(* IEC 61131-3 sources: MotionTestBenchMaster/Logical/30_MC/Libraries/MotionLib/FB, 9 files *)

(* ---- FB_AbsolutePosCalculation.st ---- *)
FUNCTION_BLOCK FB_AbsolutePosCalculation
	IF i_xEnable THEN

		IF NOT i_pstAxis.iq_stStatus.q_stMainAxisStatus.q_xInitDone OR i_pstAxis.iq_stStatus.q_stMainAxisStatus.q_xError THEN
			xPositionValid 		:= FALSE;
		ELSIF i_xPositionSensor AND NOT xPositionValid THEN
			lrAbsolutePosition 	:= i_pstAxis.iq_stStatus.q_stMainAxisStatus.q_lrPosition + 360.0 * MAX((i_uiAbsolutePositionOffset - 1), 0);
			xPositionValid 		:= TRUE;
			lrOldPosition 		:= i_pstAxis.iq_stStatus.q_stMainAxisStatus.q_lrPosition;
		ELSE
			lrIncrement			:= i_pstAxis.iq_stStatus.q_stMainAxisStatus.q_lrPosition - lrOldPosition;

			IF lrIncrement < -180.0 THEN
				lrIncrement := lrIncrement + 360.0;
			ELSIF lrIncrement > 180.0 THEN
				lrIncrement := lrIncrement - 360.0;
			END_IF

			lrAbsolutePosition	:= lrAbsolutePosition + lrIncrement;
			lrOldPosition		:= i_pstAxis.iq_stStatus.q_stMainAxisStatus.q_lrPosition;
		END_IF

		lrAbsolutePosition		:= FC_LongRealReminder(lrAbsolutePosition, 360.0 * i_uiStepsNumber, 0);

		q_xPositionValid		:= xPositionValid;
		q_lrAbsolutePosition	:= lrAbsolutePosition;
	END_IF
END_FUNCTION_BLOCK

(* ---- FB_CamGenerator.st ---- *)
(* Cam Generator Function Block *)
FUNCTION_BLOCK FB_CamGenerator
	IF i_xEnable AND i_usiNumberOfPulse > 0 THEN
		IF i_usiNumberOfPulse = 1 AND i_rOnPosition <> i_rOffPosition THEN
			rAdvPosition		:= i_rAdvanceTime * i_prAxisVelocity / 1000.0;
			q_xAdvError			:= (ABS(rAdvPosition) >= 360);

			i_pxPointerStepAdv	:= ((i_rOnPosition - rAdvPosition) < 0);

			rOnPositionA		:= FC_RealReminder(i_rOnPosition - rAdvPosition,	360.0, 0);
			rOffPositionA		:= FC_RealReminder(i_rOffPosition - rAdvPosition,	360.0, 0);

			(* CAM A GENERATION *)
			IF(rOnPositionA < rOffPositionA) THEN
				xCamValueA	:= (i_plrAxisPosition >= rOnPositionA) AND (i_plrAxisPosition < rOffPositionA);
			ELSE
				xCamValueA	:= i_plrAxisPosition >= rOnPositionA OR i_plrAxisPosition < rOffPositionA;
			END_IF

			IF xCamValueA <> xOldCamValueA THEN
				rTempReal	:= SEL(xCamValueA, rOffPositionA, rOnPositionA);
				rTempReal	:= rTempReal - LREAL_TO_REAL(i_plrAxisPosition);
				IF ABS(rTempReal) > 0.5 AND ABS(rTempReal) < 359.5 THEN
					xOldCamValueA := xCamValueA;
				END_IF
			END_IF

			(* CAM B GENERATION *)
			IF i_rOnPositionB <> 0 AND i_rOffPositionB <> 0 THEN
				rOnPositionB		:= FC_RealReminder(i_rOnPositionB - rAdvPosition,	360.0, 0);
				rOffPositionB		:= FC_RealReminder(i_rOffPositionB - rAdvPosition,	360.0, 0);
				IF(rOnPositionB < rOffPositionB) THEN
					xCamValueB	:= (i_plrAxisPosition >= rOnPositionB) AND (i_plrAxisPosition < rOffPositionB);
				ELSE
					xCamValueB	:= i_plrAxisPosition >= rOnPositionB OR i_plrAxisPosition < rOffPositionB;
				END_IF

				IF xCamValueB <> xOldCamValueB THEN
					rTempReal	:= SEL(xCamValueB, rOffPositionB, rOnPositionB);
					rTempReal	:= rTempReal - LREAL_TO_REAL(i_plrAxisPosition);
					IF ABS(rTempReal) > 0.5 AND ABS(rTempReal) < 359.5 THEN
						xOldCamValueB	:=	xCamValueB;
					END_IF
				END_IF

				(* Debounce *)
				CASE usiStep OF
					0:(* INIT *)
						usiStep := 100;

					100:(* WAIT FOR CAM A RAISING EDGE *)
						IF xCamValueA THEN
							i_pxPointerOutput := TRUE;
							usiStep := 110;
						END_IF

					110:(* WAIT FOR CAM B FALLING EDGE *)
						IF NOT xCamValueB THEN
							usiStep := 120;
						END_IF

					120:(*  WAIT FOR CAM A FALLING EDGE *)
						IF NOT xCamValueA THEN
							i_pxPointerOutput := FALSE;
							usiStep := 130;
						END_IF

					130:(* WAIT FOR CAM B RAISING EDGE *)
						IF xCamValueB THEN
							usiStep := 100;
						END_IF

					ELSE
						usiStep := 200;
				END_CASE
			ELSE
				(* Simple cam A generator *)
				i_pxPointerOutput	:= xOldCamValueA;
			END_IF
		ELSIF i_usiNumberOfPulse <= 10 THEN
			i_pxPointerStepAdv	:= FALSE;
			i_pxPointerOutput	:= FC_RealReminder(LREAL_TO_REAL(i_plrAxisPosition), 360.0 / i_usiNumberOfPulse, 0) >= 180.0 / i_usiNumberOfPulse;
		END_IF
	ELSE
		i_pxPointerOutput	:= FALSE;
		q_xAdvError			:= FALSE;
	END_IF
END_FUNCTION_BLOCK

(* Cam Generator Function Block *)
FUNCTION_BLOCK FB_CamGenerator_v2
	IF i_xEnable AND i_usiNumberOfPulse > 0 THEN
		IF i_usiNumberOfPulse = 1 AND i_rOnPosition <> i_rOffPosition THEN
			rPosition			:= DINT_TO_REAL(i_pdiAxisPosition MOD 36000) / 100.0;
			rAdvPosition		:= i_rAdvanceTime * i_prAxisVelocity / 100000.0; //v1.4
			q_xAdvError			:= (ABS(rAdvPosition) >= 360);

			i_pxPointerStepAdv	:= ((i_rOnPosition - rAdvPosition) < 0);

			rOnPosition		:= FC_RealReminder(i_rOnPosition - rAdvPosition,	360.0, 0);
			rOffPosition	:= FC_RealReminder(i_rOffPosition - rAdvPosition,	360.0, 0);

			(* CAM GENERATION *)
			IF(rOnPosition < rOffPosition) THEN
				xCamValue	:= (rPosition >= rOnPosition) AND (rPosition < rOffPosition);
			ELSE
				xCamValue	:= rPosition >= rOnPosition OR rPosition < rOffPosition;
			END_IF

			IF xCamValue <> xOldCamValue THEN
				rTempReal	:= SEL(xCamValue, rOffPosition, rOnPosition);
				rTempReal	:= rTempReal - rPosition;
				IF ABS(rTempReal) > 0.5 AND ABS(rTempReal) < 359.5 THEN
					xOldCamValue := xCamValue;
				END_IF
			END_IF

			i_pxPointerOutput	:= xOldCamValue;
		ELSIF i_usiNumberOfPulse <= 10 THEN
			i_pxPointerStepAdv	:= FALSE;
			rPosition			:= DINT_TO_REAL(i_pdiAxisPosition MOD 36000) / 100.0;
			i_pxPointerOutput	:= FC_RealReminder(rPosition, 360.0 / i_usiNumberOfPulse, 0) >= 180.0 / i_usiNumberOfPulse;
		END_IF
	ELSE
		i_pxPointerOutput	:= FALSE;
		q_xAdvError			:= FALSE;
	END_IF
END_FUNCTION_BLOCK

(* ---- FB_CamGeneratorAB.st ---- *)
(* Cam Generator Function Block *)
FUNCTION_BLOCK FB_CamGeneratorAB
	IF i_xEnable THEN
		IF (i_rOnPositionA <> i_rOffPositionA) AND (i_rOnPositionB <> i_rOffPositionB) THEN
			rAdvPosition		:= i_rAdvanceTime * i_prAxisVelocity / 1000.0;
			q_xAdvError			:= (ABS(rAdvPosition) >= 360);

			i_pxPointerStepAdvA	:= ((i_rOnPositionA - rAdvPosition) < 0);
			i_pxPointerStepAdvB	:= ((i_rOnPositionB - rAdvPosition) < 0);

			rOnPositionA		:= FC_RealReminder(i_rOnPositionA - rAdvPosition,	360.0, 0);
			rOffPositionA		:= FC_RealReminder(i_rOffPositionA - rAdvPosition,	360.0, 0);

			rOnPositionB		:= FC_RealReminder(i_rOnPositionB - rAdvPosition,	360.0, 0);
			rOffPositionB		:= FC_RealReminder(i_rOffPositionB - rAdvPosition,	360.0, 0);

			(* CAM A GENERATION *)
			IF(rOnPositionA < rOffPositionA) THEN
				xCamValueA	:= (i_plrAxisPosition >= rOnPositionA) AND (i_plrAxisPosition < rOffPositionA);
			ELSE
				xCamValueA	:= i_plrAxisPosition >= rOnPositionA OR i_plrAxisPosition < rOffPositionA;
			END_IF

			IF xCamValueA <> xOldCamValueA THEN
				rTempReal	:= SEL(xCamValueA, rOffPositionA, rOnPositionA);
				rTempReal	:= rTempReal - LREAL_TO_REAL(i_plrAxisPosition);
				IF ABS(rTempReal) > 0.5 AND ABS(rTempReal) < 359.5 THEN
					xOldCamValueA := xCamValueA;
				END_IF
			END_IF

			(* CAM B GENERATION *)
			IF(rOnPositionB < rOffPositionB) THEN
				xCamValueB	:= (i_plrAxisPosition >= rOnPositionB) AND (i_plrAxisPosition < rOffPositionB);
			ELSE
				xCamValueB	:= i_plrAxisPosition >= rOnPositionB OR i_plrAxisPosition < rOffPositionB;
			END_IF

			IF xCamValueB <> xOldCamValueB THEN
				rTempReal	:= SEL(xCamValueB, rOffPositionB, rOnPositionB);
				rTempReal	:= rTempReal - LREAL_TO_REAL(i_plrAxisPosition);
				IF ABS(rTempReal) > 0.5 AND ABS(rTempReal) < 359.5 THEN
					xOldCamValueB	:=	xCamValueB;
				END_IF
			END_IF

			(* Debounce *)
			CASE usiStep OF
				0:(* INIT *)
					usiStep := 10;

				10:(* WAIT FIRST CAM RAISING EDGE *)
					IF rOnPositionB < rOffPositionA THEN
						IF xCamValueA THEN
							i_pxPointerOutputA := TRUE;
							usiStep := 100;
						END_IF
					ELSE
						IF xCamValueB THEN
							i_pxPointerOutputB := TRUE;
							usiStep := 200;
						END_IF
					END_IF

				100:(* WAIT CAM B RISE EDGE *)
					IF xCamValueB THEN
						i_pxPointerOutputB := TRUE;
						usiStep := 110;
					END_IF

				110:(* WAIT CAM A FALLING EDGE *)
					IF NOT xCamValueA THEN
						i_pxPointerOutputA := FALSE;
						usiStep := 120;
					END_IF

				120:(* WAIT FOR CAM B FALLING EDGE *)
					IF NOT xCamValueB THEN
						i_pxPointerOutputB := FALSE;
						usiStep := 10;
					END_IF

				200:(* WAIT CAM A RISE EDGE *)
					IF xCamValueA THEN
						i_pxPointerOutputA := TRUE;
						usiStep := 210;
					END_IF

				210:(* WAIT CAM B FALLING EDGE *)
					IF NOT xCamValueB THEN
						i_pxPointerOutputB := FALSE;
						usiStep := 220;
					END_IF

				220:(* WAIT FOR CAM A FALLING EDGE *)
					IF NOT xCamValueA THEN
						i_pxPointerOutputA := FALSE;
						usiStep := 10;
					END_IF

				ELSE
					usiStep := 255;
			END_CASE
		END_IF
	ELSE
		i_pxPointerOutputA	:= FALSE;
		i_pxPointerOutputB	:= FALSE;
		q_xAdvError			:= FALSE;
	END_IF
END_FUNCTION_BLOCK

(* Cam Generator Function Block *)
FUNCTION_BLOCK FB_CamGeneratorAB_v2
	IF i_xEnable THEN
		IF (i_rOnPositionA <> i_rOffPositionA) AND (i_rOnPositionB <> i_rOffPositionB) THEN
			rPosition			:= DINT_TO_REAL(i_pdiAxisPosition MOD 36000) / 100.0;
			rAdvPosition		:= i_rAdvanceTime * i_prAxisVelocity / 100000.0; //v1.6
			q_xAdvError			:= (ABS(rAdvPosition) >= 360);

			i_pxPointerStepAdvA	:= ((i_rOnPositionA - rAdvPosition) < 0);
			i_pxPointerStepAdvB	:= ((i_rOnPositionB - rAdvPosition) < 0);

			rOnPositionA		:= FC_RealReminder(i_rOnPositionA - rAdvPosition,	360.0, 0);
			rOffPositionA		:= FC_RealReminder(i_rOffPositionA - rAdvPosition,	360.0, 0);

			rOnPositionB		:= FC_RealReminder(i_rOnPositionB - rAdvPosition,	360.0, 0);
			rOffPositionB		:= FC_RealReminder(i_rOffPositionB - rAdvPosition,	360.0, 0);

			(* CAM A GENERATION *)
			IF(rOnPositionA < rOffPositionA) THEN
				xCamValueA	:= (rPosition >= rOnPositionA) AND (rPosition < rOffPositionA);
			ELSE
				xCamValueA	:= rPosition >= rOnPositionA OR rPosition < rOffPositionA;
			END_IF

			IF xCamValueA <> xOldCamValueA THEN
				rTempReal	:= SEL(xCamValueA, rOffPositionA, rOnPositionA);
				rTempReal	:= rTempReal - rPosition;
				IF ABS(rTempReal) > 0.5 AND ABS(rTempReal) < 359.5 THEN
					xOldCamValueA := xCamValueA;
				END_IF
			END_IF

			(* CAM B GENERATION *)
			IF(rOnPositionB < rOffPositionB) THEN
				xCamValueB	:= (rPosition >= rOnPositionB) AND (rPosition < rOffPositionB);
			ELSE
				xCamValueB	:= rPosition >= rOnPositionB OR rPosition < rOffPositionB;
			END_IF

			IF xCamValueB <> xOldCamValueB THEN
				rTempReal	:= SEL(xCamValueB, rOffPositionB, rOnPositionB);
				rTempReal	:= rTempReal - rPosition;
				IF ABS(rTempReal) > 0.5 AND ABS(rTempReal) < 359.5 THEN
					xOldCamValueB	:=	xCamValueB;
				END_IF
			END_IF

			(* Debounce *)
			CASE usiStep OF
				0:(* INIT *)
					usiStep := 10;

				10:(* WAIT FIRST CAM RAISING EDGE *)
					IF rOnPositionB < rOffPositionA THEN
						IF xCamValueA THEN
							i_pxPointerOutputA := TRUE;
							usiStep := 100;
						END_IF
					ELSE
						IF xCamValueB THEN
							i_pxPointerOutputB := TRUE;
							usiStep := 200;
						END_IF
					END_IF

				100:(* WAIT CAM B RISE EDGE *)
					IF xCamValueB THEN
						i_pxPointerOutputB := TRUE;
						usiStep := 110;
					END_IF

				110:(* WAIT CAM A FALLING EDGE *)
					IF NOT xCamValueA THEN
						i_pxPointerOutputA := FALSE;
						usiStep := 120;
					END_IF

				120:(* WAIT FOR CAM B FALLING EDGE *)
					IF NOT xCamValueB THEN
						i_pxPointerOutputB := FALSE;
						usiStep := 10;
					END_IF

				200:(* WAIT CAM A RISE EDGE *)
					IF xCamValueA THEN
						i_pxPointerOutputA := TRUE;
						usiStep := 210;
					END_IF

				210:(* WAIT CAM B FALLING EDGE *)
					IF NOT xCamValueB THEN
						i_pxPointerOutputB := FALSE;
						usiStep := 220;
					END_IF

				220:(* WAIT FOR CAM A FALLING EDGE *)
					IF NOT xCamValueA THEN
						i_pxPointerOutputA := FALSE;
						usiStep := 10;
					END_IF

				ELSE
					usiStep := 255;
			END_CASE
		END_IF
	ELSE
		i_pxPointerOutputA	:= FALSE;
		i_pxPointerOutputB	:= FALSE;
		q_xAdvError			:= FALSE;
	END_IF
END_FUNCTION_BLOCK

(* ---- FB_DigitalCam.st ---- *)
FUNCTION_BLOCK FB_DigitalCam
	IF i_rOnCam > 360.0 OR i_rOnCam < 0.0 OR i_rOffCam > 360.0 OR i_rOffCam < 0.0 THEN
		uiMngStep	:= 9999;
	END_IF

	IF ((i_rOnCam = i_rOffCam) AND (i_usiPulses <= 1)) OR (i_usiPulses = 0) THEN
		uiMngStep := 0;
	END_IF

	IF i_pstAxis.move.mode <> ncPAR_LIST_MOVE AND uiMngStep = 100 AND fbCamSwitch.Enable THEN
		uiMngStep := 10;
	END_IF

	CASE uiMngStep OF
		0: 	(* Idle - Check parameters consistation *)
			fbCamSwitch.InitTrackOptions	:= FALSE;
			fbCamSwitch.Enable				:= FALSE;

			IF (i_rOnCam <> i_rOffCam) OR (i_usiPulses > 1) THEN
				uiMngStep := 100;
				stMasterSwitch.Master	:= ADR(i_pstAxis);
				stMasterSwitch.Period 	:= 360.0;
			END_IF

		10:
			fbCamSwitch.InitTrackOptions	:= FALSE;
			fbCamSwitch.Enable				:= FALSE;

			IF i_pstAxis.move.mode = ncPAR_LIST_MOVE THEN
				uiMngStep := 100;
				fbCamSwitch.Enable	:= TRUE;
			END_IF

		100:
			IF EDGEPOS(i_xRefreshClock) THEN
				IF usiMultiPulse <> i_usiPulses THEN
					uiMngStep := 600;
				ELSIF usiMultiPulse = 1 THEN
					IF stMasterSwitch.MasterStartPosition = 0.0 THEN
						IF (i_rOnCam <> stMasterSwitch.Switches[0].FirstOnPosition[0]) OR
							(i_rOffCam <> stMasterSwitch.Switches[0].LastOnPosition[0]) THEN
							stMasterSwitch.Switches[0].FirstOnPosition[0]	:= i_rOnCam;
							stMasterSwitch.Switches[0].LastOnPosition[0]	:= i_rOffCam;
							uiMngStep := 500;
						END_IF
					ELSE
						IF (i_rOnCam <> stMasterSwitch.MasterStartPosition) OR
							(i_rOffCam <> (stMasterSwitch.Switches[0].LastOnPosition[0] - (360.0 - stMasterSwitch.MasterStartPosition))) THEN
							stMasterSwitch.Switches[0].FirstOnPosition[0]	:= i_rOnCam;
							stMasterSwitch.Switches[0].LastOnPosition[0]	:= i_rOffCam;
							uiMngStep := 500;
						END_IF
					END_IF
				ELSIF i_rAdvTime <> (stTrackOption.OnCompensation * 1000.0) THEN
					uiMngStep := 400;
				END_IF
			END_IF

		400:
			stTrackOption.OnCompensation	:= i_rAdvTime / 1000.0;
			stTrackOption.OffCompensation	:= i_rAdvTime / 1000.0;
			fbCamSwitch.InitTrackOptions	:= TRUE;
			uiMngStep := 410;

		410:
			IF fbCamSwitch.TrackOptionsInitialized THEN
				fbCamSwitch.InitTrackOptions	:= FALSE;
				uiMngStep := 100;
			END_IF

		500:	(* Check parameters consistation *)
			IF stMasterSwitch.Switches[0].FirstOnPosition[0] < stMasterSwitch.Switches[0].LastOnPosition[0] THEN
				uiMngStep := 700;
			ELSE
				uiMngStep := 800;
			END_IF

		600:
			FOR usiTemp := 0 TO MAX(usiMultiPulse, i_usiPulses) - 1 DO
				IF usiTemp <= i_usiPulses - 1 THEN
					IF usiTemp = 0 THEN
						stMasterSwitch.Switches[0].FirstOnPosition[usiTemp]	:= 0.0;
						stMasterSwitch.Switches[0].LastOnPosition[usiTemp]	:= 180.0 / USINT_TO_REAL(i_usiPulses);
					ELSE
						stMasterSwitch.Switches[0].FirstOnPosition[usiTemp]	:= stMasterSwitch.Switches[0].LastOnPosition[0] * USINT_TO_REAL(usiTemp * 2);
						stMasterSwitch.Switches[0].LastOnPosition[usiTemp]	:= stMasterSwitch.Switches[0].LastOnPosition[0] * (USINT_TO_REAL(usiTemp * 2) + 1.0);
					END_IF
				ELSE
					stMasterSwitch.Switches[0].FirstOnPosition[usiTemp]	:= 0.0;
					stMasterSwitch.Switches[0].LastOnPosition[usiTemp]	:= 0.0;
				END_IF
			END_FOR

			usiMultiPulse := i_usiPulses;
			stMasterSwitch.MasterStartPosition	:= 0.0;
			stTrackOption.OnCompensation		:= i_rAdvTime / 1000.0;
			stTrackOption.OffCompensation		:= i_rAdvTime / 1000.0;
			uiMngStep := 2000;

		700:	(* Init switch 4 *)
			stMasterSwitch.MasterStartPosition	:= 0.0;
			stTrackOption.OnCompensation		:= i_rAdvTime / 1000.0;
			stTrackOption.OffCompensation		:= i_rAdvTime / 1000.0;
			uiMngStep := 2000;

		800:
			stMasterSwitch.MasterStartPosition				:= stMasterSwitch.Switches[0].FirstOnPosition[0];
			stMasterSwitch.Switches[0].LastOnPosition[0]	:= stMasterSwitch.Switches[0].LastOnPosition[0] + (360.0 - stMasterSwitch.Switches[0].FirstOnPosition[0]);
			stMasterSwitch.Switches[0].FirstOnPosition[0]	:= 0.0;
			stTrackOption.OnCompensation					:= i_rAdvTime / 1000.0;
			stTrackOption.OffCompensation					:= i_rAdvTime / 1000.0;
			uiMngStep := 2000;

		2000:
			IF EDGENEG(fbCamSwitch.Value) OR NOT fbCamSwitch.Enable THEN
				fbCamSwitch.Enable	:= FALSE;
				uiMngStep		:= 2010;
			END_IF

		2010:
			IF NOT fbCamSwitch.InOperation THEN
				fbCamSwitch.Enable	:= TRUE;
				uiMngStep		:= 2020;
			END_IF

		2020:
			IF NOT fbCamSwitch.Error AND fbCamSwitch.InOperation THEN
				uiMngStep := 100;
				xCamInitialized := TRUE;
			END_IF

		9999:
			IF NOT(i_rOnCam > 360.0 OR i_rOnCam > 0.0 OR i_rOffCam > 360.0 OR i_rOffCam > 0.0) THEN
				uiMngStep	:= 0;
			END_IF
	END_CASE

	fbCamSwitch(
	Switches		:= stMasterSwitch,
	OutputOptions	:= stOutputOption,
	TrackOptions	:= stTrackOption,
	EnableValue		:= TRUE,
	);

	q_xOutPulse := fbCamSwitch.Value;
END_FUNCTION_BLOCK

(* ---- FB_EncEmul.st ---- *)
(*********************************************************************************
 * Copyright:
 * Author:    		EncoderEmulationManagement
 * Created:  		July 4, 2016/2:37 PM
 * HELP REFERENCE:  ncsoftware/acp10_drivefunctions/acp10_drivefunctions-63-15.html
 *********************************************************************************)

(* Encoder Emulation on 8BAC130.001-1 plug-in module*)
FUNCTION_BLOCK FB_EncEmul
	IF i_pstEncEmulAxis.nc_obj_inf.node_nr > 0 AND i_pstEncEmulAxis.network.phase  <> 90 AND uiStep > 0 THEN
		uiStep := 950;
	ELSIF fbAxisError.Error	THEN
		uiStep := 960;
	ELSIF fbAxisError.Enable AND (fbAxisError.FunctionBlockErrorCount > 0 OR fbAxisError.AxisErrorCount > 0 ) THEN
		uiStep := 970;
	END_IF

	CASE uiStep OF
		0:(* DISABLE *)
			q_xError 					:= FALSE;
			q_xActive					:= FALSE;
			fbReadParID.Execute 		:= FALSE;
			fbWriteParID_Text.Execute 	:= FALSE;
			fbWriteParID.Execute 		:= FALSE;

			IF NOT i_xErrorReset AND i_pstEncEmulAxis.network.phase  = 90 AND i_pstEncEmulAxis.nc_obj_inf.node_nr > 0 THEN
				fbAxisError.Axis	:= ADR(i_pstEncEmulAxis);
				fbAxisError.Mode	:= mcNO_TEXT + mcACKNOWLEDGE_ALL;
				fbAxisError.Enable	:= TRUE; //V4.A.A.1.6.13
				uiStep				:= 10;
			END_IF

		(**************************** CONFIGURE ENCODER EMULATION ****************************)
		10:(* ENCODER TYPE CONFIG *)
			IF NOT fbWriteParID.Execute THEN
				usiTemp						:= ncINC_OUTPUT;

				fbWriteParID.Axis			:= ADR(i_pstEncEmulAxis);
				fbWriteParID.DataAddress 	:= ADR(usiTemp);
				fbWriteParID.DataType		:= ncPAR_TYP_USINT;
				fbWriteParID.ParID			:= ACP10PAR_ENCOD_TYPE;
				fbWriteParID.Execute		:= TRUE;
			END_IF

			IF fbWriteParID.Done AND fbWriteParID.ParID = ACP10PAR_ENCOD_TYPE THEN
				fbWriteParID.Execute	:= FALSE;
				uiStep					:= 20;
			ELSIF fbWriteParID.Error THEN
				uiStep					:= 900;
			END_IF
		(* ENCODER MODE CONFIG *)
		20:(* INC MODE *)
			IF NOT fbWriteParID.Execute THEN
				uiTemp						:= 4;

				fbWriteParID.Axis			:= ADR(i_pstEncEmulAxis);
				fbWriteParID.DataAddress 	:= ADR(uiTemp);
				fbWriteParID.DataType		:= ncPAR_TYP_UINT;
				fbWriteParID.ParID			:= ACP10PAR_ENCOD_INC_MODE;
				fbWriteParID.Execute		:= TRUE;
			END_IF

			IF fbWriteParID.Done AND fbWriteParID.ParID = ACP10PAR_ENCOD_INC_MODE THEN
				fbWriteParID.Execute	:= FALSE;
				uiStep					:= 30;
			ELSIF fbWriteParID.Error THEN
				uiStep					:= 900;
			END_IF

		30:(* SCALE ENC INCREMENT CONFIG *)
			IF NOT fbWriteParID.Execute THEN
				udiTemp						:= UINT_TO_UDINT(i_uiNumberOfPulses) * 64;

				fbWriteParID.Axis			:= ADR(i_pstEncEmulAxis);
				fbWriteParID.DataAddress 	:= ADR(udiTemp);
				fbWriteParID.DataType		:= ncPAR_TYP_UDINT;
				fbWriteParID.ParID			:= ACP10PAR_SCALE_ENCOD_INCR;
				fbWriteParID.Execute		:= TRUE;
			END_IF

			IF fbWriteParID.Done AND fbWriteParID.ParID = ACP10PAR_SCALE_ENCOD_INCR THEN
				fbWriteParID.Execute	:= FALSE;
				uiStep					:= 40;
			ELSIF fbWriteParID.Error THEN
				uiStep					:= 900;
			END_IF

		40:(* SCALE LOAD UNITS CONFIG *)
			IF NOT fbWriteParID.Execute THEN
				udiTemp						:= 36000;

				fbWriteParID.Axis			:= ADR(i_pstEncEmulAxis);
				fbWriteParID.DataAddress 	:= ADR(udiTemp);
				fbWriteParID.DataType		:= ncPAR_TYP_UDINT;
				fbWriteParID.ParID			:= ACP10PAR_SCALE_LOAD_UNITS;
				fbWriteParID.Execute		:= TRUE;
			END_IF

			IF fbWriteParID.Done AND fbWriteParID.ParID = ACP10PAR_SCALE_LOAD_UNITS THEN
				fbWriteParID.Execute	:= FALSE;
				IF i_pstSrcAxis.nc_obj_inf.node_nr = i_pstEncEmulAxis.nc_obj_inf.node_nr THEN
					uiStep := 200;		//CONFIGURE CROSSLINK
				ELSE
					uiStep := 100;		//CONFIGURE NETWORK COUPLING
				END_IF
			ELSIF fbWriteParID.Error THEN
				uiStep := 900;
			END_IF

		(************************** CONFIGURE NETWORK COUPLING ******************************)
		100:(* Sender config: MA3_CYCLIC_SEND <- PCTRL_S_SET / S_VAX1 *)
			IF NOT fbWriteParID.Execute THEN
				IF i_pstSrcAxis.nc_obj_inf.nc_obj_typ = ncAXIS THEN
					uiTemp		:= ACP10PAR_PCTRL_S_SET; 	//REAL AXIS
				ELSE
					uiTemp		:= ACP10PAR_S_SET_VAX1;		//VIRTUAL AXIS
				END_IF

				fbWriteParID.Axis			:= ADR(i_pstSrcAxis);
				fbWriteParID.DataAddress 	:= ADR(uiTemp);
				fbWriteParID.DataType		:= ncPAR_TYP_UINT;
				fbWriteParID.ParID			:= ACP10PAR_MA3_CYCLIC_SEND;
				fbWriteParID.Execute		:= TRUE;
			END_IF

			IF fbWriteParID.Done AND fbWriteParID.ParID = ACP10PAR_MA3_CYCLIC_SEND THEN
				fbWriteParID.Execute	:= FALSE;
				uiStep					:= 120;
			ELSIF fbWriteParID.Error THEN
				uiStep					:= 900;
			END_IF

		120:(* Receiver config : MA5_CYCLIC_POS <- "node_nr [+ 256 for AXIS 2], MA3_CYCLIC_SEND" *)
			IF NOT fbWriteParID_Text.Execute THEN
				uiTemp		:= i_pstSrcAxis.nc_obj_inf.node_nr + 256 * (i_pstSrcAxis.nc_obj_inf.nc_obj_idx);
				itoa(uiTemp, ADR(strTemp));
				uiTemp		:= ACP10PAR_MA3_CYCLIC_SEND;
				itoa(uiTemp, ADR(strTemp2));

				strcat(ADR(strTemp), ADR(', '));
				strcat(ADR(strTemp), ADR(strTemp2));

				fbWriteParID_Text.Axis			:= ADR(i_pstEncEmulAxis);
				fbWriteParID_Text.DataText	 	:= strTemp;
				fbWriteParID_Text.ParID			:= ACP10PAR_CONFIG_MA5_CYCLIC_POS;
				fbWriteParID_Text.Execute		:= TRUE;
			END_IF

			IF fbWriteParID_Text.Done AND fbWriteParID_Text.ParID = ACP10PAR_CONFIG_MA5_CYCLIC_POS THEN
				fbWriteParID_Text.Execute	:= FALSE;
				uiStep						:= 140;
			ELSIF fbWriteParID_Text.Error THEN
				uiStep					:= 900;
			END_IF

		140:(* Set interpolation mode = LINEAR *)
			IF NOT fbWriteParID.Execute THEN
				usiTemp						:= 1;	//LINEAR MODE

				fbWriteParID.Axis			:= ADR(i_pstEncEmulAxis);
				fbWriteParID.DataAddress 	:= ADR(usiTemp);
				fbWriteParID.DataType		:= ncPAR_TYP_USINT;
				fbWriteParID.ParID			:= ACP10PAR_MA5_CYCLIC_IPL_MODE;
				fbWriteParID.Execute		:= TRUE;
			END_IF

			IF fbWriteParID.Done AND fbWriteParID.ParID = ACP10PAR_MA5_CYCLIC_IPL_MODE THEN
				fbWriteParID.Execute	:= FALSE;
				uiStep					:= 150;
			ELSIF fbWriteParID.Error THEN
				uiStep					:= 900;
			END_IF

		150:(* CHECK COMMUNICATION STATUS *)
			IF NOT fbReadParID.Execute THEN
				fbReadParID.Axis			:= ADR(i_pstEncEmulAxis);
				fbReadParID.DataAddress 	:= ADR(usiErrCode);
				fbReadParID.DataType		:= ncPAR_TYP_USINT;
				fbReadParID.ParID			:= ACP10PAR_MA5_CYCLIC_ERROR_STATUS;
				fbReadParID.Execute			:= TRUE;
			END_IF

			IF fbReadParID.Done AND fbReadParID.ParID = ACP10PAR_MA5_CYCLIC_ERROR_STATUS THEN
				fbReadParID.Execute	:= FALSE;
				IF usiErrCode = ERR_OK THEN
					uiEncodOutParID		:= ACP10PAR_MA5_CYCLIC_POS;
					IF i_xEnable THEN
						uiStep	:= 250;
					ELSE
						uiStep	:= 400;
					END_IF
				ELSE
					uiStep				:= 800;
				END_IF
			ELSIF fbReadParID.Error THEN
				uiStep					:= 900;
			END_IF

		(**************************** CONFIGURE CROSSLINK ****************************)
		200:(* CONFIGURE CROSSLINK SOURCE AXIS *)
			IF NOT fbWriteParID.Execute THEN
				uiTemp						:= i_pstSrcAxis.nc_obj_inf.nc_obj_idx + 1;

				fbWriteParID.Axis			:= ADR(i_pstEncEmulAxis);
				fbWriteParID.DataAddress 	:= ADR(uiTemp);
				fbWriteParID.DataType		:= ncPAR_TYP_UINT;
				fbWriteParID.ParID			:= ACP10PAR_CROSSLINK_AXIS;
				fbWriteParID.Execute		:= TRUE;
			END_IF

			IF fbWriteParID.Done AND fbWriteParID.ParID = ACP10PAR_CROSSLINK_AXIS THEN
				fbWriteParID.Execute	:= FALSE;
				uiStep					:= 210;
			ELSIF fbWriteParID.Error THEN
				uiStep					:= 900;
			END_IF

		210:(* CONFIGURE CROSSLINK PARID <- PCTRL_S_SET / S_SET_VAX1 *)
			IF NOT fbWriteParID.Execute THEN
				IF i_pstSrcAxis.nc_obj_inf.nc_obj_typ = ncAXIS THEN
					uiTemp		:= ACP10PAR_PCTRL_S_SET;	//REAL AXIS
				ELSE
					uiTemp		:= ACP10PAR_S_SET_VAX1;		//VIRTUAL AXIS
				END_IF

				fbWriteParID.Axis			:= ADR(i_pstEncEmulAxis);
				fbWriteParID.DataAddress 	:= ADR(uiTemp);
				fbWriteParID.DataType		:= ncPAR_TYP_UINT;
				fbWriteParID.ParID			:= ACP10PAR_CROSSLINK_PARID;
				fbWriteParID.Execute		:= TRUE;
			END_IF

			IF fbWriteParID.Done AND fbWriteParID.ParID = ACP10PAR_CROSSLINK_PARID THEN
				fbWriteParID.Execute	:= FALSE;
				uiEncodOutParID			:= ACP10PAR_CROSSLINK_PARID;
				IF i_xEnable THEN
					uiStep	:= 250;
				ELSE
					uiStep	:= 400;
				END_IF
			ELSIF fbWriteParID.Error THEN
				uiStep					:= 900;
			END_IF

		250:(* ENABLE ENCODER EMULATOR OUTPUT *)
			IF NOT fbWriteParID.Execute THEN
				fbWriteParID.Axis			:= ADR(i_pstEncEmulAxis);
				fbWriteParID.DataAddress 	:= ADR(uiEncodOutParID);
				fbWriteParID.DataType		:= ncPAR_TYP_UINT;
				fbWriteParID.ParID			:= ACP10PAR_ENCOD_OUT_PARID;
				fbWriteParID.Execute		:= TRUE;
			END_IF

			IF fbWriteParID.Done AND fbWriteParID.ParID = ACP10PAR_ENCOD_OUT_PARID THEN
				fbWriteParID.Execute	:= FALSE;
				uiStep					:= 300;
			ELSIF fbWriteParID.Error THEN
				uiStep					:= 900;
			END_IF

		300:(* READY *)
			fbAxisError.Enable	:= TRUE;
			q_xActive			:= TRUE;

			IF NOT i_xEnable THEN
				uiStep			:= 400;
			END_IF

		400:(* DISABLE OUTPUT *)
			//fbAxisError.Enable	:= FALSE; //V4.A.A.1.6.13

			IF NOT fbWriteParID.Execute THEN
				uiTemp						:= 0;

				fbWriteParID.Axis			:= ADR(i_pstEncEmulAxis);
				fbWriteParID.DataAddress 	:= ADR(uiTemp);
				fbWriteParID.DataType		:= ncPAR_TYP_UINT;
				fbWriteParID.ParID			:= ACP10PAR_ENCOD_OUT_PARID;
				fbWriteParID.Execute		:= TRUE;
			END_IF

			IF fbWriteParID.Done AND fbWriteParID.ParID = ACP10PAR_ENCOD_OUT_PARID THEN
				fbWriteParID.Execute	:= FALSE;
				q_xActive 				:= FALSE;
				uiStep	:= 410;
			END_IF

		410: (* OUTPUT DISABLED *)
			IF i_xEnable THEN
				uiStep	:= 250;
			END_IF

		(********************************************)
		800:(* CYCLIC COMMUNICATION ERROR *)
			q_xError 		:= TRUE;
			q_uiErrorID		:= usiErrCode;
			IF i_xErrorReset THEN
				q_xError 	:= FALSE;
				q_uiErrorID := 0;
				uiStep		:= 0;
			END_IF

		900:(* FUNCTION BLOCKS ERROR *)
			q_xError 		:= TRUE;
			q_uiErrorID 	:= fbWriteParID.ErrorID + fbReadParID.ErrorID + fbWriteParID_Text.ErrorID;

			fbWriteParID.Execute 	:= FALSE;
			fbReadParID.Execute 	:= FALSE;

			IF i_xErrorReset THEN
				IF fbWriteParID.Error THEN
					fbWriteParID.Execute := FALSE;
				END_IF
				IF fbReadParID.Error THEN
					fbReadParID.Execute := FALSE;
				END_IF
				IF fbWriteParID_Text.Error THEN
					fbReadParID.Execute := FALSE;
				END_IF
			END_IF

			IF NOT fbWriteParID.Error AND NOT fbReadParID.Error AND NOT fbWriteParID_Text.Error THEN
				q_xError 		:= FALSE;
				q_uiErrorID 	:= 0;
				uiStep			:= 0;
			END_IF

		950:
			fbWriteParID.Execute 	:= FALSE;
			fbReadParID.Execute 	:= FALSE;

			q_xError 		:= TRUE;
			q_uiErrorID		:= 60000;
			IF i_pstEncEmulAxis.network.phase  = 90 THEN
				uiStep	:= 0;
			END_IF

		960:
			fbWriteParID.Execute 	:= FALSE;
			fbReadParID.Execute 	:= FALSE;

			q_xError 	:= TRUE;
			q_uiErrorID	:= 60010;

			IF i_xErrorReset THEN
				fbAxisError.Enable	:= FALSE;
			END_IF

			IF NOT fbAxisError.Error THEN
				uiStep	:= 0;
			END_IF

		970:
			q_xError 	:= TRUE;
			q_uiErrorID	:= 60020;

			fbWriteParID.Execute 	:= FALSE;
			fbReadParID.Execute 	:= FALSE;

			//fbAxisError.Acknowledge	:= i_xErrorReset; //V4.A.A.1.6.13

			IF NOT(fbAxisError.FunctionBlockErrorCount > 0 OR fbAxisError.AxisErrorCount > 0) THEN
				//fbAxisError.Enable	:= FALSE; //V4.A.A.1.6.13
				uiStep	:= 0;
			END_IF
	END_CASE

	(* Acknowledge Error *)
	fbAxisError.Acknowledge	:= i_xErrorReset;

	fbAxisError();
	fbReadParID();
	fbWriteParID_Text();
	fbWriteParID();
END_FUNCTION_BLOCK

(* ---- FB_ExceptionAlarmX.st ---- *)
(* Fb for mananging alarms *)
FUNCTION_BLOCK FB_ExceptionAlarmX
	IF i_pxInitCoreDone THEN
		IF i_xConditions AND NOT xAlarmActive THEN
			xAlarmActive := TRUE;
			MpAlarmXSet(MpLink := i_pstMpAlarmXLink, Name := i_psAlarmName);
		ELSIF NOT i_xConditions AND xAlarmActive THEN
			IF i_pxAcknowledge OR i_xAutoAck THEN
				xAlarmActive := FALSE;
				MpAlarmXReset(MpLink := i_pstMpAlarmXLink, Name := i_psAlarmName);
			END_IF
		END_IF
		q_xAlarmActive := xAlarmActive;
	END_IF
END_FUNCTION_BLOCK

(* ---- FB_Periodic2ContinuePosition.st ---- *)
FUNCTION_BLOCK FB_Periodic2ContinuePosition
	IF NOT i_xEnable THEN
		xActive 		:= FALSE;
		diOldInPosition := 0;
		q_diPosition	:= 0;
		RETURN;
	ELSIF NOT xActive THEN
		xActive 		:= TRUE;
		q_diPosition	:= i_diInPosition;
		diOldInPosition := i_diInPosition;
	ELSE
		(* Continue DINT position calculation *)
		IF ABS(i_diInPosition - diOldInPosition) < UDINT_TO_DINT(i_udiPeriod / 2) THEN
			q_diPosition		:= q_diPosition + (i_diInPosition - diOldInPosition);
		ELSIF i_diInPosition < diOldInPosition THEN
			q_diPosition		:= q_diPosition + i_udiPeriod + (i_diInPosition - diOldInPosition);
		ELSE
			q_diPosition		:= q_diPosition - i_udiPeriod + (i_diInPosition - diOldInPosition);
		END_IF
		diOldInPosition 	:= i_diInPosition;
	END_IF
END_FUNCTION_BLOCK

(* ---- FB_Position2Velocity.st ---- *)
FUNCTION_BLOCK FB_Position2Velocity
	fbRTInfo(enable := TRUE);
	adiBuffer[uiCount]	:= i_diPosition;
	IF uiCount > 0 THEN
		arBufferVel[uiCount] := DINT_TO_REAL((i_diPosition - adiBuffer[uiCount - 1])) / (DINT_TO_REAL(fbRTInfo.cycle_time) * 1E-6);
	ELSE
		arBufferVel[uiCount] := DINT_TO_REAL((i_diPosition - adiBuffer[c_usiNSample - 1])) / (DINT_TO_REAL(fbRTInfo.cycle_time) * 1E-6);
	END_IF

	uiCount 	:= (uiCount + 1) MOD c_usiNSample;
	rInternal	:= 0;

	FOR i := 0 TO c_usiNSample - 1 DO
		rInternal	:= rInternal + arBufferVel[i];
	END_FOR

	q_rVelocity := rInternal / c_usiNSample;
END_FUNCTION_BLOCK

(* ---- FB_Step2PeriodicPosition.st ---- *)
(* From a step signal a periodic signal is created *)
FUNCTION_BLOCK FB_PeriodicPosition
	IF NOT i_xEnable OR i_rPeriod <=0 THEN
		usiStep				:= 0;
		q_xPositionValid	:= FALSE;
	ELSE
		CASE usiStep OF
			0:
				q_xPositionValid	:= FALSE;
				q_rPeriodicPosition	:= 0;
				rPosition			:= 0;

				IF i_xEnable THEN
					usiStep	:= 10;
				END_IF

			10:
				IF EDGEPOS(i_xResetPostion) THEN
					q_xPositionValid	:= TRUE;
					rPosition			:= i_rAxisPosition;
					q_rPeriodicPosition	:= i_rAxisPosition;
					usiStep				:= 20;
				END_IF

			20:
				rDeltaPos	:= i_rAxisPosition - rPosition;
				// If the difference between the old axis and the current axis position
				// If greater than 180° it means that we overlapped the period
				IF ABS(rDeltaPos) > 180 THEN
					IF rDeltaPos > 0 THEN
						rDeltaPos	:= rDeltaPos - 360;
					ELSE
						rDeltaPos	:= rDeltaPos + 360;
					END_IF
				END_IF

				q_rPeriodicPosition	:= FC_RealReminder(q_rPeriodicPosition + rDeltaPos, i_rPeriod, 0);
				rPosition			:= i_rAxisPosition;

				IF i_xResetPostion	THEN
					usiStep	:= 0;
				END_IF
		END_CASE
	END_IF
END_FUNCTION_BLOCK
